// TIA Portal V19 export
DATA_BLOCK "AI SCALING DB"   // DB5
{ S7_Optimized_Access := 'FALSE' }
   VAR RETAIN
      SET : Struct
         "OXIDATION REDUCTION POTENTIO METER 301" : Int;
         "CONDUCTIVITY INDUCTOR CUM TRANSMITTER 301" : Int;
         "PH INDICATOR CUM TRANSMITTER 301" : Int;
         "PH INDICATOR CUM TRANSMITTER 302" : Int;
         "CONDUCTIVITY INDICATOR CUM TRANSMITTER 302" : Int;
         "LEVEL TRANSMITTER 401" : Int;
         "PH INDICATOR CUM TRANSMITTER 401" : Int;
         "CONDUCTIVITY INDICATOR CUM TRANSMITTER 401" : Int;
         "CONFUCTIVITY INDICATOR CUM TRANSMITTER 402" : Int;
         "PH INDICATOR CUM TRANSMITTER 402" : Int;
         "LEVEL TRANSMITTER 501" : Int;
         "FLOW INDICATOR TOTALOZER 501" : Int;
         "PRESSURE TRANSMITTER 501" : Int;
         "FLOW INDICATOR TRANSMITTER 502" : Int;
         "PRESSURE TRANSMITTER 502" : Int;
         "PRESSURE TRANSMITTER 503" : Int;
         "PRESSURE TRANSMITTER 504" : Int;
         "PRESSURE TRANSMITTER 505" : Int;
         "PRESSURE TRANSMITTER 506" : Int;
         "PH INDICATOR CUM TRANSMITTER 501" : Int;
         "PH INDICATOR CUM TRANSMITTER 502" : Int;
         "RESISTIVITY CUM TRANSMITTER 501" : Int;
         "RESISTIVITY CUM TRANSMITTER 502" : Int;
         "LEVEL TRANSMITTER 502" : Int;
         "FLOW INDICATOR TRANSMITTER 503" : Int;
         "FLOW INDICATOR TRANSMITTER 504" : Int;
         "FLOW INDICATOR TRANSMITTER 505" : Int;
         "FLOW INDICATOR TRANSMITTER 506" : Int;
         "FLOW INDICATOR TRANSMITTER 507" : Int;
         "FLOW INDICATOR TRANSMITTER 508" : Int;
         "SPARE(6)" : Int;
         "SPARE(7)" : Int;
      END_STRUCT;
      MIN : Struct
         "OXIDATION REDUCTION POTENTIO METER 301" { S7_SetPoint := 'True'} : Real := -1900.0;
         "CONDUCTIVITY INDUCTOR CUM TRANSMITTER 301" { S7_SetPoint := 'True'} : Real;
         "PH INDICATOR CUM TRANSMITTER 301" { S7_SetPoint := 'True'} : Real;
         "PH INDICATOR CUM TRANSMITTER 302" { S7_SetPoint := 'True'} : Real;
         "CONDUCTIVITY INDICATOR CUM TRANSMITTER 302" { S7_SetPoint := 'True'} : Real;
         "LEVEL TRANSMITTER 401" { S7_SetPoint := 'True'} : Real;
         "PH INDICATOR CUM TRANSMITTER 401" { S7_SetPoint := 'True'} : Real;
         "CONDUCTIVITY INDICATOR CUM TRANSMITTER 401" { S7_SetPoint := 'True'} : Real;
         "CONFUCTIVITY INDICATOR CUM TRANSMITTER 402" { S7_SetPoint := 'True'} : Real;
         "PH INDICATOR CUM TRANSMITTER 402" { S7_SetPoint := 'True'} : Real;
         "LEVEL TRANSMITTER 501" { S7_SetPoint := 'True'} : Real;
         "FLOW INDICATOR TOTALOZER 501" { S7_SetPoint := 'True'} : Real;
         "PRESSURE TRANSMITTER 501" { S7_SetPoint := 'True'} : Real;
         "FLOW INDICATOR TRANSMITTER 502" { S7_SetPoint := 'True'} : Real;
         "PRESSURE TRANSMITTER 502" : Real;
         "PRESSURE TRANSMITTER 503" : Real;
         "PRESSURE TRANSMITTER 504" : Real;
         "PRESSURE TRANSMITTER 505" : Real;
         "PRESSURE TRANSMITTER 506" : Real;
         "PH INDICATOR CUM TRANSMITTER 501" : Real;
         "PH INDICATOR CUM TRANSMITTER 502" : Real;
         "RESISTIVITY CUM TRANSMITTER 501" : Real;
         "RESISTIVITY CUM TRANSMITTER 502" : Real;
         "LEVEL TRANSMITTER 502" : Real;
         "FLOW INDICATOR TRANSMITTER 503" : Real;
         "FLOW INDICATOR TRANSMITTER 504" : Real;
         "FLOW INDICATOR TRANSMITTER 505" : Real;
         "FLOW INDICATOR TRANSMITTER 506" : Real;
         "FLOW INDICATOR TRANSMITTER 507" : Real;
         "FLOW INDICATOR TRANSMITTER 508" : Real;
         "SPARE(6)" : Real;
         "SPARE(7)" : Real;
      END_STRUCT;
      MAX : Struct
         "OXIDATION REDUCTION POTENTIO METER 301" { S7_SetPoint := 'True'} : Real := 1900.0;
         "CONDUCTIVITY INDUCTOR CUM TRANSMITTER 301" { S7_SetPoint := 'True'} : Real := 1999.0;
         "PH INDICATOR CUM TRANSMITTER 301" { S7_SetPoint := 'True'} : Real := 14.0;
         "PH INDICATOR CUM TRANSMITTER 302" { S7_SetPoint := 'True'} : Real := 14.0;
         "CONDUCTIVITY INDICATOR CUM TRANSMITTER 302" { S7_SetPoint := 'True'} : Real := 1999.0;
         "LEVEL TRANSMITTER 401" { S7_SetPoint := 'True'} : Real := 100.0;
         "PH INDICATOR CUM TRANSMITTER 401" { S7_SetPoint := 'True'} : Real := 14.0;
         "CONDUCTIVITY INDICATOR CUM TRANSMITTER 401" { S7_SetPoint := 'True'} : Real := 1999.0;
         "CONFUCTIVITY INDICATOR CUM TRANSMITTER 402" { S7_SetPoint := 'True'} : Real := 1999.0;
         "PH INDICATOR CUM TRANSMITTER 402" { S7_SetPoint := 'True'} : Real := 14.0;
         "LEVEL TRANSMITTER 501" { S7_SetPoint := 'True'} : Real := 100.0;
         "FLOW INDICATOR TOTALOZER 501" { S7_SetPoint := 'True'} : Real := 14.0;
         "PRESSURE TRANSMITTER 501" { S7_SetPoint := 'True'} : Real := 6.0;
         "FLOW INDICATOR TRANSMITTER 502" { S7_SetPoint := 'True'} : Real := 14.0;
         "PRESSURE TRANSMITTER 502" { S7_SetPoint := 'True'} : Real := 6.0;
         "PRESSURE TRANSMITTER 503" { S7_SetPoint := 'True'} : Real := 6.0;
         "PRESSURE TRANSMITTER 504" { S7_SetPoint := 'True'} : Real := 6.0;
         "PRESSURE TRANSMITTER 505" { S7_SetPoint := 'True'} : Real := 6.0;
         "PRESSURE TRANSMITTER 506" { S7_SetPoint := 'True'} : Real := 6.0;
         "PH INDICATOR CUM TRANSMITTER 501" { S7_SetPoint := 'True'} : Real := 14.0;
         "PH INDICATOR CUM TRANSMITTER 502" { S7_SetPoint := 'True'} : Real := 14.0;
         "RESISTIVITY CUM TRANSMITTER 501" { S7_SetPoint := 'True'} : Real := 100.0;
         "RESISTIVITY CUM TRANSMITTER 502" { S7_SetPoint := 'True'} : Real := 100.0;
         "LEVEL TRANSMITTER 502" { S7_SetPoint := 'True'} : Real := 100.0;
         "FLOW INDICATOR TRANSMITTER 503" { S7_SetPoint := 'True'} : Real := 5.0;
         "FLOW INDICATOR TRANSMITTER 504" { S7_SetPoint := 'True'} : Real := 5.0;
         "FLOW INDICATOR TRANSMITTER 505" { S7_SetPoint := 'True'} : Real := 1000.0;
         "FLOW INDICATOR TRANSMITTER 506" { S7_SetPoint := 'True'} : Real := 150.0;
         "FLOW INDICATOR TRANSMITTER 507" { S7_SetPoint := 'True'} : Real := 150.0;
         "FLOW INDICATOR TRANSMITTER 508" { S7_SetPoint := 'True'} : Real := 1000.0;
         "SPARE(6)" { S7_SetPoint := 'True'} : Real;
         "SPARE(7)" : Real;
      END_STRUCT;
      PV : Struct
         "OXIDATION REDUCTION POTENTIO METER 301" : Real;
         "CONDUCTIVITY INDUCTOR CUM TRANSMITTER 301" : Real;
         "PH INDICATOR CUM TRANSMITTER 301" : Real;
         "PH INDICATOR CUM TRANSMITTER 302" : Real;
         "CONDUCTIVITY INDICATOR CUM TRANSMITTER 302" : Real;
         "LEVEL TRANSMITTER 401" : Real;
         "PH INDICATOR CUM TRANSMITTER 401" : Real;
         "CONDUCTIVITY INDICATOR CUM TRANSMITTER 401" : Real;
         "CONFUCTIVITY INDICATOR CUM TRANSMITTER 402" : Real;
         "PH INDICATOR CUM TRANSMITTER 402" : Real;
         "LEVEL TRANSMITTER 501" : Real;
         "FLOW INDICATOR TOTALOZER 501" : Real;
         "PRESSURE TRANSMITTER 501" : Real;
         "FLOW INDICATOR TRANSMITTER 502" : Real;
         "PRESSURE TRANSMITTER 502" : Real;
         "PRESSURE TRANSMITTER 503" : Real;
         "PRESSURE TRANSMITTER 504" : Real;
         "PRESSURE TRANSMITTER 505" : Real;
         "PRESSURE TRANSMITTER 506" : Real;
         "PH INDICATOR CUM TRANSMITTER 501" : Real;
         "PH INDICATOR CUM TRANSMITTER 502" : Real;
         "RESISTIVITY CUM TRANSMITTER 501" : Real;
         "RESISTIVITY CUM TRANSMITTER 502" : Real;
         "LEVEL TRANSMITTER 502" : Real;
         "FLOW INDICATOR TRANSMITTER 503" : Real;
         "FLOW INDICATOR TRANSMITTER 504" : Real;
         "FLOW INDICATOR TRANSMITTER 505" : Real;
         "FLOW INDICATOR TRANSMITTER 506" : Real;
         "FLOW INDICATOR TRANSMITTER 507" : Real;
         "FLOW INDICATOR TRANSMITTER 508" : Real;
         "SPARE(6)" : Real;
         "SPARE(7)" : Real;
      END_STRUCT;
      SPARE : Bool;
      SPARE_1 : Bool;
      "LT-401" : Struct
         LOW_BUFF : Int;
         HIGH_BUFF : Int;
      END_STRUCT;
      "LT-501" : Struct
         LOW_BUFF : Int;
         HIGH_BUFF : Int;
      END_STRUCT;
      "LT-502" : Struct
         LOW_BUFF : Int;
         HIGH_BUFF : Int;
      END_STRUCT;
      "LT-401 SET VALVE" : Struct
         LL : Real;
         L : Real;
         H : Real;
         HH : Real;
      END_STRUCT;
      "LT-501 SET VALVE" : Struct
         LL : Real;
         L : Real;
         H : Real;
         HH : Real;
      END_STRUCT;
      "LT-502 SET VALVE" : Struct
         LL : Real;
         L : Real;
         H : Real;
         HH : Real;
      END_STRUCT;
   END_VAR
BEGIN
END_DATA_BLOCK
